{attribute addProperty BoxType "EL2262--0000"}
{attribute addProperty Id "Cycle_CounterAT %Q*Cycle_Counter_485675001620Sample_0AT %Q*Sample_2F9FC35D810WcStateAT %I*WcState_64F6A8C6810InfoDataAT %I*InfoData_7231B2DD80100"}
{attribute addProperty CRC "1794052630"}
{attribute addProperty SizeInBites "112"}
{attribute addProperty SizeInBytes "14"}
TYPE EL2262_CED6AB5C :
STRUCT
	{attribute addProperty Name "Cycle_Counter"}
	Cycle_Counter : Cycle_Counter_48567500;
	{attribute addProperty Name "Sample_0"}
	Sample_0 : Sample_2F9FC35D;
	{attribute addProperty Name "WcState"}
	WcState : WcState_64F6A8C6;
	{attribute addProperty Name "InfoData"}
	InfoData : InfoData_7231B2DD;
END_STRUCT
END_TYPE

(* stored: Version 1.2.0.0, ProductVersion 3.1.4024.9
   DUT EL2262_CED6AB5C: Id {9f546d23-9a1a-4cf0-a34a-febe1080c2a4} *)
